{attribute 'GeneratedUsingTerminal: '}
{attribute addProperty BoxType ""}
{attribute addProperty Id "unreferencedAT %I*SyncUnitTask_2D604ED59PlcTaskAT %I*SyncUnitTask_2D604ED59"}
{attribute addProperty CRC "1877705303"}
{attribute addProperty Size "18"}
TYPE SyncUnitTasks_6FEB8257 :
STRUCT
	{attribute addProperty Name "unreferenced"}
	unreferenced : SyncUnitTask_2D604ED5;
	{attribute addProperty Name "PlcTask"}
	PlcTask : SyncUnitTask_2D604ED5;
END_STRUCT
END_TYPE

(* stored: Version 1.2.0.0, ProductVersion 3.1.4024.9
   DUT SyncUnitTasks_6FEB8257: Id {dc4a45f8-6eec-4a7d-8e7f-c2cf688c0cf2} *)
